FUNCTION_BLOCK F_ADD (* Adds two number values *)
  PACKAGE iec61131::arithmetic;
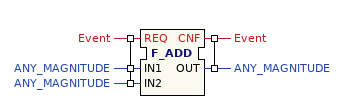
  EVENT_INPUT
    REQ WITH IN1, IN2; (* Normal Execution Request *)
  END_EVENT
  EVENT_OUTPUT
    CNF WITH OUT; (* Execution Confirmation *)
  END_EVENT
  VAR_INPUT
    IN1 : ANY_MAGNITUDE; (* First funtion input *)
    IN2 : ANY_MAGNITUDE; (* Second function input *)
  END_VAR
  VAR_OUTPUT
    OUT : ANY_MAGNITUDE; (* IN1 plus IN2 *)
  END_VAR
END_FUNCTION_BLOCK
